INTERFACE I_DIGroup

// Add input to group
METHOD AddInput
VAR_INPUT
	IDI			: I_DigitalIn;		// Interface to digital input
END_VAR
END_METHOD

// Gets the total number of IOs in the group
PROPERTY Count : INT
GET
END_GET
END_PROPERTY

// Determine the command from the inputs in the group
METHOD GetCommand : E_DICommand
END_METHOD

// Get a specific input from the group
METHOD GetInput : I_DigitalIn
VAR_INPUT
	nInputIndex		: INT;		// Input index
END_VAR
END_METHOD

// Set input group mode (default OR)
PROPERTY Mode : E_DIGroupMode
SET
END_SET
END_PROPERTY

END_INTERFACE

(* stored: Version 1.1.0.1, ProductVersion 3.1.4024.12
   Itf I_DIGroup: Id {47af0e41-2432-4a87-a436-53179529a67a}
   Folder Methods: Id {994b8b7d-16c0-4a44-9f40-a832e8ed5871}
   Folder Properties: Id {7635148f-1bc0-4447-8062-31dd6668195d}
   Method AddInput: Id {e5d7ee1b-ab47-422d-9ca9-d608d338ffbd}
   Property Count: Id {04300eab-0eb0-45f6-897c-5d3b70ee1a7e}
   Get Get: Id {92cfac21-00b3-4f30-80f2-7f54689eada7}
   Method GetCommand: Id {6320d08d-1fef-473b-a8e4-8266b5d5899c}
   Method GetInput: Id {15dc0faf-d9f3-49bb-8df8-bf91dcd02d4e}
   Property Mode: Id {82d1dade-437a-4999-b446-d332f2876426}
   Set Set: Id {f311e281-f2a1-4c71-a07e-8e99f812e526} *)
